Staubli VAL3: pickNplaceShelf.pgx

program pickNplaceShelf()
begin
  //assumption : arm in cal_ref1

  //pick f1
  //wait until user confirm (reload bottom
  //place f1
  //pick f2
  //wait until user confirm (close the fixture
  //place f2 (need blow simultanously
  //pick f3
  //place f3

end
